TYPE ST_ServiceStatus :
STRUCT
	ResponseId : UDINT;
	PackMLOut : ST_PML_Base_Out;
	ExecuteSubState : ST_ServiceExecuteSubStateStatus;
	CompletionBehavior : E_ServiceCompletionBehavior;
	ServiceId : UDINT;
	ErrorList : ARRAY[1..Param_Config.MaxServiceError] OF ST_ExtAlarm;
	Data : ST_ServiceDataStatus;
END_STRUCT
END_TYPE

(* stored: Version 1.1.0.1, ProductVersion 3.1.4026.18
   DUT ST_ServiceStatus: Id {696bda33-0a33-48b0-8ccd-362e4a358520} *)
